(* PLC project FBDExample.project, CODESYS CODESYS V3.5 SP14 Patch 1 *)
(* stored: creationDateTime 2019-02-25T11:45:43.3471801, modificationDateTime 2019-02-22T15:27:06.5143224 *)

FUNCTION_BLOCK FBD1
  VAR_INPUT
    a : BOOL;
    b : BOOL;
    c : BOOL;
  END_VAR
  VAR_OUTPUT
    x : BOOL;
    y : BOOL;
    z : BOOL;
    o : INT;
  END_VAR
  VAR
    i : INT;
    j : INT;
    k : INT;
  END_VAR
  VAR  (* added by the conversion: wires and edge detectors of the diagram *)
    _SUB10000000004_OUT : INT;
    _ADD10000000008_OUT : INT;
    _MUX10000000012_OUT : INT;
    _EXECUTE20000000004_EN : BOOL;
    _OR20000000007_OUT : BOOL;
  END_VAR

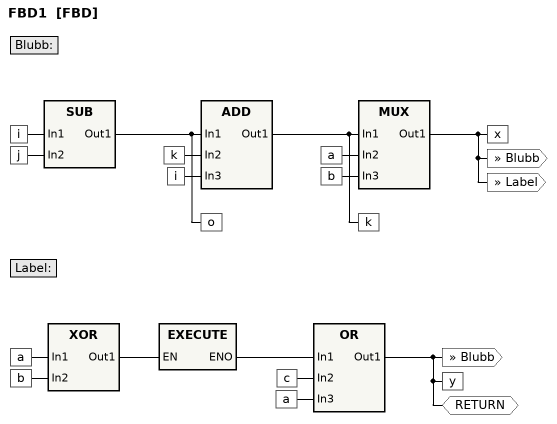
(* FBD diagram, written out as Structured Text *)
Blubb:
_SUB10000000004_OUT := i - j;
o := _SUB10000000004_OUT;
_ADD10000000008_OUT := _SUB10000000004_OUT + k + i;
k := _ADD10000000008_OUT;
_MUX10000000012_OUT := MUX(_ADD10000000008_OUT, a, b);
x := _MUX10000000012_OUT;
IF _MUX10000000012_OUT THEN JMP Blubb; END_IF;
IF _MUX10000000012_OUT THEN JMP Label; END_IF;
Label:
_EXECUTE20000000004_EN := a XOR b;
IF _EXECUTE20000000004_EN THEN
  x:= x AND x;
END_IF;
_OR20000000007_OUT := _EXECUTE20000000004_EN OR c OR a;
IF _OR20000000007_OUT THEN JMP Blubb; END_IF;
y := _OR20000000007_OUT;
IF _OR20000000007_OUT THEN RETURN; END_IF;
END_FUNCTION_BLOCK

FUNCTION_BLOCK FBDRecursive
  VAR_OUTPUT
    intern : INT;
  END_VAR
  VAR
    o : INT;
  END_VAR
  VAR  (* added by the conversion: wires and edge detectors of the diagram *)
    _ADD30000000003_OUT : INT;
  END_VAR

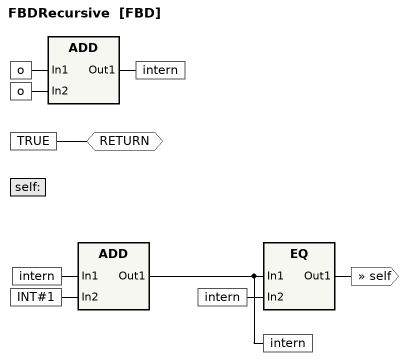
(* FBD diagram, written out as Structured Text *)
intern := o + o;
IF TRUE THEN RETURN; END_IF;
self:
_ADD30000000003_OUT := intern + INT#1;
intern := _ADD30000000003_OUT;
IF _ADD30000000003_OUT = intern THEN JMP self; END_IF;
END_FUNCTION_BLOCK

PROGRAM POU
  VAR
    f : FBD1;
    g : FBDRecursive;
  END_VAR

            g();
f();
          
END_PROGRAM
